// TIA Portal project "Ejercicio1" (V15.1)

(* hardware
DEVICE "HMI_1"  KTP700 Basic PN
   slot 0: "HMI_1"  KTP700 Basic PN  6AV2 123-2GB03-0AX0  15.1.0.0
   slot 1: "HMI_RT_1"  KTP700 Basic PN  6AV2 123-2GB03-0AX0  15.1.0.0
   slot 5: "HMI_1.IE_CP_1"  PROFINET Interface  15.0.1.0
      slot 1: "Interfaz PROFINET_1"  PROFINET Interface
         slot 1: "Port_1"  Port
DEVICE "S7-1200 station_1"  S7-1200 Station
   slot 0: "Rack_0"  S7-1200 Rack  Rack  V1.0
   slot 1: "PLC_1"  CPU 1215C AC/DC/Rly  6ES7 215-1BG40-0XB0  V4.2
*)

// ===== PLC "PLC_1"  CPU 1215C AC/DC/Rly =====

VAR_GLOBAL   // PLC tag table "Tabla de variables estándar"
   "System_Byte" AT %MB8191 : Byte;
   "FirstScan" AT %M8191.0 : Bool;
   "DiagStatusUpdate" AT %M8191.1 : Bool;
   "AlwaysTRUE" AT %M8191.2 : Bool;
   "AlwaysFALSE" AT %M8191.3 : Bool;
   "Clock_Byte" AT %MB1 : Byte;
   "Clock_10Hz" AT %M1.0 : Bool;
   "Clock_5Hz" AT %M1.1 : Bool;
   "Clock_2.5Hz" AT %M1.2 : Bool;
   "Clock_2Hz" AT %M1.3 : Bool;
   "Clock_1.25Hz" AT %M1.4 : Bool;
   "Clock_1Hz" AT %M1.5 : Bool;
   "Clock_0.625Hz" AT %M1.6 : Bool;
   "Clock_0.5Hz" AT %M1.7 : Bool;
   "Interruptor ON/OFF" AT %M0.0 : Bool;
   "Lampara de funcionamiento" AT %M10.0 : Bool;
   "Palanca de giro positivo motor" AT %M0.1 : Bool;
   "Palanca de giro negativo motor" AT %M0.2 : Bool;
   "Lampara sentido positivo giro" AT %M10.1 : Bool;
   "Lampara sentido negativo giro" AT %M10.2 : Bool;
   "Contactor giro positivo motor" AT %M10.3 : Bool;
   "Contactor giro negativo motor" AT %M10.4 : Bool;
   "Sensor de temperatura" AT %M0.3 : Bool;
   "Piloto panel de mando" AT %M10.5 : Bool;
END_VAR

ORGANIZATION_BLOCK "Main"   // OB1, LAD, ProgramCycle
TITLE = "Main Program Sweep (Cycle)"
{ S7_Optimized_Access := 'TRUE' }
VERSION : 0.1
   VAR_INPUT
      Initial_Call : Bool;   // Initial call of this OB
      Remanence : Bool;   // =True, if remanent data are available
   END_VAR
   VAR_TEMP   // added for the SCL form of the ladder/FBD networks
      _w1 : Bool;
      _w2 : Bool;
   END_VAR
BEGIN

REGION Network 1
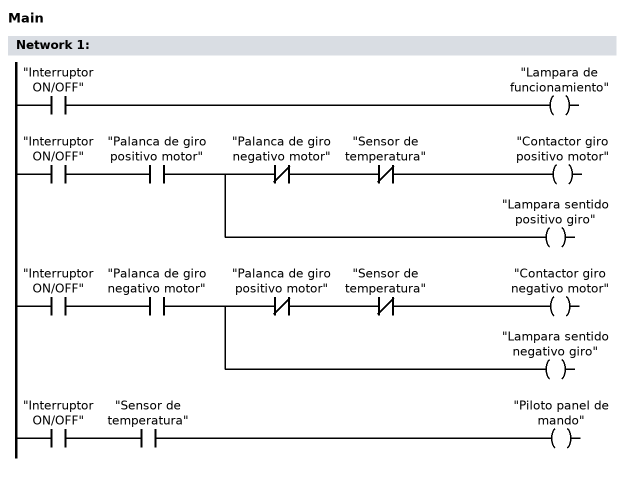
   RUNG wire#powerrail
      Contact( "Interruptor ON/OFF" )
      Coil( "Lampara de funcionamiento" )
   END_RUNG
   RUNG wire#powerrail
      Contact( "Interruptor ON/OFF" )
      Contact( "Palanca de giro positivo motor" )
      wire#w1
      I_Contact( "Palanca de giro negativo motor" )
      I_Contact( "Sensor de temperatura" )
      Coil( "Contactor giro positivo motor" )
   END_RUNG
   RUNG wire#w1
      Coil( "Lampara sentido positivo giro" )
   END_RUNG
   RUNG wire#powerrail
      Contact( "Interruptor ON/OFF" )
      Contact( "Palanca de giro negativo motor" )
      wire#w2
      I_Contact( "Palanca de giro positivo motor" )
      I_Contact( "Sensor de temperatura" )
      Coil( "Contactor giro negativo motor" )
   END_RUNG
   RUNG wire#w2
      Coil( "Lampara sentido negativo giro" )
   END_RUNG
   RUNG wire#powerrail
      Contact( "Interruptor ON/OFF" )
      Contact( "Sensor de temperatura" )
      Coil( "Piloto panel de mando" )
   END_RUNG
   // the same network as SCL:
   "Lampara de funcionamiento" := "Interruptor ON/OFF";
   #_w1 := "Interruptor ON/OFF" AND "Palanca de giro positivo motor";
   "Contactor giro positivo motor" := #_w1 AND NOT "Palanca de giro negativo motor" AND NOT "Sensor de temperatura";
   "Lampara sentido positivo giro" := #_w1;
   #_w2 := "Interruptor ON/OFF" AND "Palanca de giro negativo motor";
   "Contactor giro negativo motor" := #_w2 AND NOT "Palanca de giro positivo motor" AND NOT "Sensor de temperatura";
   "Lampara sentido negativo giro" := #_w2;
   "Piloto panel de mando" := "Interruptor ON/OFF" AND "Sensor de temperatura";
END_REGION
END_ORGANIZATION_BLOCK

(* ===== HMI "HMI_RT_1" =====
system functions are stored by id; their names below are inferred from use
connection "HMI_Conexión_1": ETHERNET, SMART_S7_1200_OMS

HMI tags "Tabla de variables estándar"
   "Número_imagen_variable" : UInt, internal
   "Interruptor ON/OFF" : Bool = PLC "Interruptor ON/OFF" AT %M0.0, 1 s
   "Lampara de funcionamiento" : Bool = PLC "Lampara de funcionamiento" AT %M10.0, 1 s
   "Palanca de giro positivo motor" : Bool = PLC "Palanca de giro positivo motor" AT %M0.1, 1 s
   "Palanca de giro negativo motor" : Bool = PLC "Palanca de giro negativo motor" AT %M0.2, 1 s
   "Lampara sentido negativo giro" : Bool = PLC "Lampara sentido negativo giro" AT %M10.2, 1 s
   "Lampara sentido positivo giro" : Bool = PLC "Lampara sentido positivo giro" AT %M10.1, 1 s
   "Piloto panel de mando" : Bool = PLC "Piloto panel de mando" AT %M10.5, 1 s
   "Contactor giro positivo motor" : Bool = PLC "Contactor giro positivo motor" AT %M10.3, 1 s
   "Contactor giro negativo motor" : Bool = PLC "Contactor giro negativo motor" AT %M10.4, 1 s

text list "Nombre_imagen_lista_texto": 1 'Imagen raíz'

Template "Plantilla_1" 800x480
   Button "Salir" at 714,429 size 71x50; TextOff 'Salir'; PictureOff "ExitRuntime_KTP700_Basic_PN_TR"; PictureOn "ExitRuntime_KTP700_Basic_PN_TR"
      on Release: StopRuntime(0)
   Button "Template_Button" at 614,429 size 71x50; TextOff 'Text'
   Button "Template_Button_1" at 514,429 size 71x50; TextOff 'Text'
   Button "Template_Button_2" at 414,429 size 71x50; TextOff 'Text'
   Button "Template_Button_3" at 314,429 size 71x50; TextOff 'Text'
   Button "Template_Button_4" at 214,429 size 71x50; TextOff 'Text'
   Button "Template_Button_5" at 114,429 size 71x50; TextOff 'Text'
   Button "Imagen inicial" at 14,429 size 71x50; TextOff 'Imagen inicial'; PictureOff "NavigateHome_KTP700_Basic_PN_TR"; PictureOn "NavigateHome_KTP700_Basic_PN_TR"
      on Release: ActivateScreen("Imagen raíz", 0)
   SymbolicIOField "Imagen_campo_ES_simbólico" at 93,9 size 600x33; TextOff '0'; TextOn '1'; TextList "Nombre_imagen_lista_texto"
      ProcessValue <- "Número_imagen_variable"
      on Change: ActivateScreenByNumber("Número_imagen_variable", 0)
   DateTimeField "HmiScreenItemData" at 695,25 size 105x25
   DateTimeField "HmiScreenItemData_1" at 695,0 size 105x25
   GraphicView "Logotipo" at 0,0 size 91x51; Picture "Logotipo de HMI_1"

screen "Imagen raíz" 800x480, template "Plantilla_1"
   on GenerateScreen: SetTag("Número_imagen_variable", 1)
   Switch "Interruptor_1" at 145,143 size 64x32; CaptionText 'Switch'; TextOff 'OFF'; TextOn 'ON'
      ProcessValue <- "Interruptor ON/OFF"
   Switch "Interruptor_2" at 209,225 size 64x32; CaptionText 'Switch'; TextOff 'OFF'; TextOn 'ON'
      ProcessValue <- "Palanca de giro positivo motor"
   Switch "Interruptor_3" at 209,305 size 64x32; CaptionText 'Switch'; TextOff 'OFF'; TextOn 'ON'
      ProcessValue <- "Palanca de giro negativo motor"
   Circle "Círculo_1" at 328,216 size 48x48
      Appearance <- "Lampara sentido positivo giro"
   Circle "Círculo_2" at 327,294 size 48x48
      Appearance <- "Lampara sentido negativo giro"
   Circle "Círculo_3" at 222,136 size 48x48
      Appearance <- "Lampara de funcionamiento"
   Circle "Círculo_4" at 525,362 size 48x48
      Appearance <- "Piloto panel de mando"
   TextField "Campo de texto_1" at 131,96 size 185x23; Text 'Interruptor Encendido'
   TextField "Campo de texto_2" at 204,201 size 70x23; Text 'Positivo'
   TextField "Campo de texto_3" at 209,282 size 78x23; Text 'Negativo'
   TextField "Campo de texto_4" at 483,342 size 138x23; Text 'Panel de control'
   Circle "Círculo_5" at 416,216 size 48x48
      Appearance <- "Contactor giro positivo motor"
   Circle "Círculo_6" at 416,294 size 48x48
      Appearance <- "Contactor giro negativo motor"
*)